KUKA KRL data list: braketestselftest.dat

&ACCESS RVP
&REL 1
&PARAM TEMPLATE = C:\KRC\Roboter\Template\ExpertVorgabe
&PARAM EDITMASK = *
DEFDAT braketestselftest PUBLIC

ENDDAT
